PROGRAM INTERNAL MAIN
VAR
	_driveTest : fbDriveTest;
END_VAR

END_PROGRAM

(* stored: Version 1.1.0.1, ProductVersion 3.1.4024.5
   POU MAIN: Id {d1e7ffc5-0e5e-40b6-83db-d6d43156a01c}, SpecialFunc None *)
